{attribute addProperty BoxType "EL9550-0010-0016"}
{attribute addProperty Id "Status_UpAT %I*Status_Up_B12359DC1620Status_UsAT %I*Status_Us_B12359DC1620WcStateAT %I*WcState_F855686C1620InfoDataAT %I*InfoData_192954DE1620"}
{attribute addProperty CRC "584321072"}
{attribute addProperty SizeInBites "64"}
{attribute addProperty SizeInBytes "8"}
TYPE EL9550_E584A12F :
STRUCT
	{attribute addProperty Name "Status_Up"}
	Status_Up : Status_Up_B12359DC;
	{attribute addProperty Name "Status_Us"}
	Status_Us : Status_Us_B12359DC;
	{attribute addProperty Name "WcState"}
	WcState : WcState_F855686C;
	{attribute addProperty Name "InfoData"}
	InfoData : InfoData_192954DE;
END_STRUCT
END_TYPE

(* stored: Version 1.2.0.0, ProductVersion 3.1.4024.9
   DUT EL9550_E584A12F: Id {02ea0f12-64c0-4279-92f6-32186ae80ddd} *)
